(* CODESYS project AppSample_UDPCom_c550.project

Project tree, tasks and I/O mapping:
  c550_UDP_Example : Controller c550, Lenze, order no. FAST Runtime, version 1.11.0.21
      settings: 0x2001:0 = c550_UDP_Example; 0x2381:1 = 0; 0x2381:2 = 0; 0x2381:3 = 0; 0x2381:5 =                                 ; 0x2381:6 =                       ; 0x2381:7 =                 ; 0x2381:8 =                                                       ; 0x2451:1 = 0; 0x2451:2 = 0; 0x2451:3 = 0; 0x2451:4 = 0; 0x2459:1 = 0; 0x2459:2 = 0; 0x245A:2 = 0; 0x245A:3 = 0; 0x245A:4 = 0; 0x245A:5 = 0; 0x245B:1 = 2; 0x245C:1 = 52; 0x2471:13 = 100; 0x2471:14 = 100; 0x2471:51 = 1; 0x2471:103 = 6; 0x247B:1 = 0; 0x2859:1 = 2; 0x2859:2 = 0; 0x2859:3 = 2; 0x2859:4 = 2; 0x2859:5 = 2; 0x285A:1 = 0; 0x5820:1 = 2; 0x5851:31 = 100; 0x5910:1 = 0; 0x5910:2 = 0; 0x5910:3 = 0; 0x5910:4 = 0; 0x5910:5 = 0; 0x5910:6 = 0; 0x5910:7 = 0;
        0x5910:8 = 0; 0x5910:9 = 0; 0x5911:1 = 1; 0x5911:2 = 0; 0x5911:3 = 2; 0x5911:31 = 0; 0x5911:32 = 0; 0x5911:33 = 0; 0x5911:51 = 1; 0x5911:52 = 0; 0x5911:53 = 2; 0x5912:1 = 1; 0x5912:2 = 0; 0x5912:3 = 2; 0x5912:11 = 1; 0x5912:12 = 0; 0x5912:13 = 2; 0x5912:31 = 0; 0x5912:32 = 0; 0x5912:33 = 0; 0x5912:41 = 1; 0x5912:42 = 0; 0x5912:43 = 2; 0x5912:51 = 0; 0x5912:52 = 0; 0x5912:53 = 0; 0x5912:61 = 0; 0x5912:62 = 0; 0x5912:63 = 0; 0x5912:71 = 0; 0x5912:72 = 0; 0x5912:73 = 0; 0x5912:91 = 1; 0x5912:92 = 0; 0x5912:93 = 2; 0x5912:101 = 0; 0x5912:102 = 0; 0x5912:103 = 0; 0x5912:131 = 0; 0x5912:132 = 0;
        0x5912:133 = 0; 0x5912:151 = 0; 0x5912:152 = 0; 0x5912:153 = 0; 0x5913:1 = 0; 0x5913:2 = 0; 0x5913:3 = 0; 0x5913:7 = 0; 0x5913:8 = 50000; 0x5913:9 = 54999; 0x5913:10 = protocol name; 0x5913:11 = 0; 0x5913:12 = 0; 0x5913:13 = 0; 0x5913:17 = 0; 0x5913:18 = 50000; 0x5913:19 = 54999; 0x5913:20 = protocol name; 0x5913:21 = 0; 0x5913:22 = 0; 0x5913:23 = 0; 0x5913:27 = 0; 0x5913:28 = 50000; 0x5913:29 = 54999; 0x5913:30 = protocol name; 0x5913:31 = 0; 0x5913:32 = 0; 0x5913:33 = 0; 0x5913:37 = 0; 0x5913:38 = 50000; 0x5913:39 = 54999; 0x5913:40 = protocol name
    application Application
      libraries: CAA Types Extern, 3.5.17.0 (CAA Technical Workgroup); CAA Net Base Services, 3.5.17.0 (CAA Technical Workgroup); L_Util, 3.28.0.1 (Lenze); L_PLCLoggingAccess, 3.26.0.0 (Lenze); L_IE1P_ApplicationErrors, 3.30.0.53 (Lenze); L_MC2P_MotionControlCam, 3.30.0.17 (Lenze); L_SEMP_ErrorManagement, 3.26.0.0 (Lenze); L_IMHP_ModuleHandler, 3.30.0.11 (Lenze); L_IPAP_ParameterManagerAccess, 3.26.0.0 (Lenze); L_MC1P_MotionControlBasic, 3.30.0.173 (Lenze); L_SPMI_PlcParameterManager, 3.28.0.1 (Lenze); L_TB2P_TechModulesBasic, 3.30.0.61 (Lenze); L_TF2P_TechModulesFollowingPositioning, 3.30.0.62 (Lenze); L_TS2P_TechModulesSynchronizingCamming, 3.30.0.56 (Lenze); L_TW2P_TechModulesWindingTraversing, 3.30.0.7 (Lenze); L_TP2P_TechModulesProcessFunctions, 3.30.0.5 (Lenze); L_EtcSlaveConfig, 3.28.0.0 (Lenze); L_IC1P_ComponentDirectory, 3.30.0.8 (Lenze); L_ILMP_LicenseManager, 3.30.0.5 (Lenze); VisuDialogs, * (System)
      task MainTask (cyclic, interval t#5ms, priority 1, watchdog T#4ms x 1) calls MAIN_c550
      program MAIN_c550 [FBD]
      visualisation Visu_UDPCom_c550
      global variables GVL_ComponentHardware
      program GVL_ComponentHardwareCall [ST]
    I_O_Modul_Koppler : Coupler I/O moduls, Lenze, version 3.21.0.0
        settings: Group1 Task Name = 'MainTask'
        unmapped channels: Error, unused, unused, unused, unused, unused, unused, unused, ErrorID, AbsoluteCounter, unused, unused, unused, unused, unused, unused, unused, unused
    AxesGroups
    VirtualAxes
    ParameterEditor : Parameter Editor, Lenze, version 3.24.0.0
    FAST_System_Configuration : FAST System Configuration, Lenze, version 3.28.0.2
    FAST_System_Diagnosis : FAST System Diagnosis, Lenze, version 3.24.0.2
    OPC_UA : OPC UA Connectivity, Lenze, version 3.26.0.1
      UA_Server : OPC UA Server, Lenze, version 3.26.0.1
  text list GlobalTextList
  UDP_Com/
    function blocks/
      function block UDPCom [ST]: CreateCRC, Error, Peers, CheckIpIfBroadcastIsSet, RW
    data types/
      data type UDP_Telegram
    visualisation UDPCom_VISU
    internal/
      IpAddrHandling/
        visualisation IpAddrHandling_VISU
        FUNCTION/
          function Bytes4ToIpAddrString [ST]
          function IpAddressStringToBytes4 [ST]
        function block IpAddrHandling [ST]: CheckIpAddressSyntax
    text list NetBaseServices_ERROR
*)

// UDP_Com/data types/UDP_Telegram
{attribute 'pack_mode' := '0'}
TYPE UDP_Telegram :
STRUCT
	uiCRC: UINT; //Do not change this variable! Used for transferring the checksum!
	diUserData: DINT; //User data (can be of any type)
	//Add more user variables
END_STRUCT
END_TYPE

// c550_UDP_Example/Application/GVL_ComponentHardware
(* This code is generated automatically *)
(* Don't change the content! *)

{attribute 'qualified_only'}
{attribute 'linkalways'}
VAR_GLOBAL
	//Controller
	c550_UDP_Example 	: L_IC1P_ComponentHardware;

END_VAR

// c550_UDP_Example/Application/MAIN_c550
PROGRAM MAIN_c550
VAR
	fbUDPCom: UDPCom ;
	DataRead : UDP_Telegram;
	DataWrite: UDP_Telegram;
END_VAR

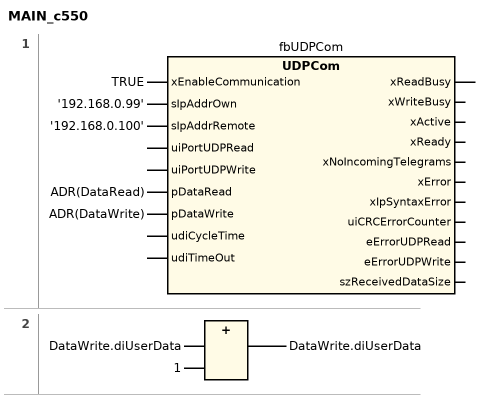
// NETWORK 1
fbUDPCom(
    xEnableCommunication := TRUE,
    sIpAddrOwn := '192.168.0.99',
    sIpAddrRemote := '192.168.0.100',
    pDataRead := ADR(DataRead),
    pDataWrite := ADR(DataWrite)); // UDPCom

// NETWORK 2
DataWrite.diUserData := DataWrite.diUserData + 1;

END_PROGRAM

// UDP_Com/function blocks/UDPCom
FUNCTION_BLOCK UDPCom
VAR_INPUT
	xEnableCommunication : BOOL;					 		  //Enabling UPD read or UPD write functions
	sIpAddrOwn			 : STRING[15];				 		  //IP address of this device
	sIpAddrRemote		 : STRING[15];				 		  //IP address of remote device
	uiPortUDPRead		 : UINT := 1240;			 		  //Port on this device via which UDP telegrams are received
	uiPortUDPWrite		 : UINT := 1241;			 		  //Port on this device via which UDP telegrams are transmitted
	pDataRead			 : POINTER TO UDP_Telegram; 		  //Passing the address of a variable of type UDP_Telegram. UDP_Telegram is a structure that contains the payload data for UDP communication
	pDataWrite			 : POINTER TO UDP_Telegram; 		  //Passing the address of a variable of type UDP_Telegram. UDP_Telegram is a structure that contains the payload data for UDP communication
	udiCycleTime		 : UDINT 					 := 100;  //Cycle time [ms] for sending UDP telegrams
	udiTimeOut			 : UDINT 					 := 2000; //Watchdog time, scaled in [ms]
END_VAR                                                   
VAR_OUTPUT                                                
	xReadBusy			 : BOOL;	   	//TRUE: Function block is busy in reading UDP data
	xWriteBusy			 : BOOL;	   	//TRUE: Function block is busy in writing UDP data
	xActive				 : BOOL;	   	//TRUE: Peers have opened for UDP communication on this device
	xReady				 : BOOL;	   	//TRUE: UDP data was read successfully
	xNoIncomingTelegrams : BOOL;	   	//TRUE: No handshake telegram has been received within the watchdog time period (udiTimeOut)
	xError				 : BOOL;	   	//TRUE: An error has occured during function block execution (for more details please refer to status output eError)
	xIpSyntaxError    	 : BOOL;	   	//TRUE: The IP address set in sIpAddrOwn and/or in sIpAddrRemote has an incorrect syntax
	uiCRCErrorCounter	 : UINT;		//If the checksum check detects incorrect data in the received telegram, uiCRCErrorCounter is incremented
	eErrorUDPRead    	 : CAA.ERROR; 	//Error number for the UDP read process, in the case of xError = TRUE
	eErrorUDPWrite	  	 : CAA.ERROR;	//Error number for the UDP write process, in the case of xError = TRUE
	szReceivedDataSize	 : CAA.SIZE;  	//Size in bytes of the received data
END_VAR
VAR
	(* FB instances *)
	fbIpAddrHandlingOwn	   : IpAddrHandling;	//Function block for IP-Address handling
	fbIpAddrHandlingRemote : IpAddrHandling;   	//Function block for IP-Address handling 	
	fbPeerRX			   : NBS.UDP_Peer;		//Function block to open a peer to read UDP telegrams on function block UDP_Receive1
	fbPeerTX			   : NBS.UDP_Peer;		//Function block to open a peer to transmit UDP telegram on function block UDP_Send1
	fbUDPReceive		   : NBS.UDP_Receive;	//Function block for reading UDP data via peer 1
	fbUDPSend			   : NBS.UDP_Send;		//Function block for transmitting UDP telegram on peer 2
	fbTrigWatchdogTimer	   : R_TRIG;    		//Edge detection to start the watchdog timer		 
	fbWatchdogTimer		   : TON;				//Timer function block for watchdog evaluation
	fbTimerCyclic		   : TON;				//Timer function block for cyclic data transmission
	
	(*Internal variables *)
	xReadActive    	: BOOL;
	xWriteActive 	: BOOL;
	szSizeDataRead 	: CAA.SIZE;
	szSizeDataWrite : CAA.SIZE;
	xBroadcastIsSet : BOOL;
	uiCRC: UINT; //CRC
END_VAR

(* Calling the block instances of IpAddrHandling ====================================================*)
fbIpAddrHandlingOwn(psIpAddrIN 		:= ADR(sIpAddrOwn));
fbIpAddrHandlingRemote(psIpAddrIN 	:= ADR(sIpAddrRemote));

xBroadcastIsSet := CheckIpIfBroadcastIsSet(sIpAddrString := sIpAddrRemote);

(* Set xIpSyntaxError ===============================================================================*)
IF fbIpAddrHandlingOwn.xIpSyntaxError OR fbIpAddrHandlingRemote.xIpSyntaxError THEN
	xIpSyntaxError := TRUE;
ELSE
	xIpSyntaxError := FALSE;
END_IF

(* Get the number of bytes of user data by dereferencing the pointer ================================*)
szSizeDataRead := SIZEOF(pDataRead^);
szSizeDataWrite := SIZEOF(pDataWrite^);

(* UDP peers ========================================================================================*)
Peers();

(* UDP read write ===================================================================================*)
RW();

(* Set errors =======================================================================================*)
Error();

(* Set output variables =============================================================================*)
xActive := xReadActive AND xWriteActive;

(* Create a simple checksum by adding a maximum of 128 byte packets *)
METHOD PRIVATE CreateCRC : UINT
VAR_INPUT
	pData: POINTER TO UDP_Telegram;
END_VAR
VAR
	paby	: POINTER TO ARRAY[0..130] OF BYTE;
	uiSize	: UINT;
	ui 		: UINT := 2;
END_VAR

paby := pData;
uiSize := SIZEOF(pData^) - 2;
IF uiSize >= 128 THEN
	uiSize := 128;
END_IF

FOR ui := 2 TO uiSize BY 1 DO
	CreateCRC := CreateCRC + paby^[ui];
END_FOR
END_METHOD

ACTION Error:
(* Set errors =======================================================================================*)

xError := fbPeerRX.xError OR fbUDPReceive.xError OR fbPeerTX.xError OR fbUDPSend.xError;

IF fbPeerRX.xError THEN        
	eErrorUDPRead := fbPeerRX.eError;
ELSIF fbUDPReceive.xError THEN  
	eErrorUDPRead := fbUDPReceive.eError;
ELSE                                
	eErrorUDPRead := 0;
END_IF

IF fbPeerTX.xError THEN
	eErrorUDPWrite := fbPeerTX.eError;
ELSIF fbUDPSend.xError THEN
	eErrorUDPWrite := fbUDPSend.eError;
ELSE
	eErrorUDPWrite := 0;
END_IF
END_ACTION

ACTION Peers:
(* READ | Open a peer to read data from remote IP address============================================*)
//Change IP-Address setting if an broadcast IP is set
IF xBroadcastIsSet THEN
	fbPeerRX.ipAddr.sAddr := sIpAddrRemote;	//setting remote IP address (access of element of structure NBS.IP_ADDR)
ELSE
	fbPeerRX.ipAddr.sAddr := sIpAddrOwn; 	//setting own IP address (access of element of structure NBS.IP_ADDR)
END_IF

//Open a peer for receive Data
fbPeerRX(xEnable := xEnableCommunication, uiPort := uiPortUDPRead);

//Set xReadActive if the peer opened successfully
xReadActive := fbPeerRX.xActive AND fbPeerRX.hPeer<>0;


(* WRITE | Open a peer to transmit data to remote IP address=========================================*)
//Open a peer for transmit Data
fbPeerTX.ipAddr.sAddr := sIpAddrOwn; // setting own IP address (access of element of structure NBS.IP_ADDR)
fbPeerTX(xEnable := xEnableCommunication, uiPort := uiPortUDPWrite);

//Set xWriteActive if the peer opened successfully
xWriteActive := fbPeerTX.xActive AND fbPeerTX.hPeer<>0;
END_ACTION

(* Check whether the last octet in the IP address is set to 255 (broadcast) *)
METHOD PRIVATE CheckIpIfBroadcastIsSet : BOOL
VAR_INPUT
	sIpAddrString: STRING[15];
END_VAR
VAR
	usiStringLengh: USINT;
	sTemp: STRING[4];
END_VAR

usiStringLengh := TO_USINT(LEN(sIpAddrString));
sTemp := MID(sIpAddrString, 4, usiStringLengh - 3);

IF sTemp = '.255' THEN
	CheckIpIfBroadcastIsSet := TRUE;
ELSE
	CheckIpIfBroadcastIsSet := FALSE;
END_IF
END_METHOD

ACTION RW:

(* READ =============================================================================================*)
//UDP receive
fbUDPReceive(xEnable := xReadActive,
			 hPeer	 := fbPeerRX.hPeer,
			 szSize	 := szSizeDataRead,
			 pData	 := pDataRead,
			 xDone	 => ,
			 xBusy	 => xReadBusy,
			 xReady	 => xReady);

//CRC check
	uiCRC := CreateCRC(pData := pDataRead);
	IF uiCRC <> pDataRead^.uiCRC THEN
		uiCRCErrorCounter := uiCRCErrorCounter + 1;
	ELSIF xEnableCommunication = FALSE THEN
		uiCRCErrorCounter := 0;
	END_IF
	
//Get number of bytes received from the sender
IF fbUDPReceive.xReady OR NOT xReadActive THEN
	szReceivedDataSize := fbUDPReceive.szCount; 
END_IF

//Generation of watchdog alert
fbTrigWatchdogTimer(CLK	:= xReady);
fbWatchdogTimer(IN	:= xReadActive AND NOT fbTrigWatchdogTimer.Q AND (udiTimeOut<>0),
				PT	:= UDINT_TO_TIME(udiTimeOut),
				Q	=> xNoIncomingTelegrams);

(* WRITE ============================================================================================*)
//Logic for cyclic transmission
fbTimerCyclic(IN := NOT fbTimerCyclic.Q, PT	:= UDINT_TO_TIME(LIMIT(9,udiCycleTime-1,4294967294))); 

//Execute UDP transmission
fbUDPSend.xExecute := xWriteActive AND (udiCycleTime > 0 AND fbTimerCyclic.Q); 

//Create CRC
IF fbUDPSend.xExecute THEN
	pDataWrite^.uiCRC := CreateCRC(pData := pDataWrite);
END_IF

//UDP send
fbUDPSend.ipAddr.sAddr	:= sIpAddrRemote; 
fbUDPSend(	hPeer 	:= fbPeerTX.hPeer,
			uiPort	:= uiPortUDPWrite,
			szSize	:= szSizeDataWrite,
			pData	:= pDataWrite,	
			xDone	=> ,				
			xBusy	=> );
END_ACTION

END_FUNCTION_BLOCK

// UDP_Com/internal/IpAddrHandling/IpAddrHandling
(*	This function block is responsible for setting an IP address. This can be changed in two places:												*)
(*		1. In a user-created variable of type STRING[15]. To do this, 																				*)
(*		   the address of this variable must be transferred to the function block input “psIpAddrIN”.												*)
(*		2. In the visualization "IpAddrHandling_VISU" available for this function block.															*)
(*																																					*)
(*	If the address is changed with correct syntax in one of these two places, it is output in "sIpAddrOut". If the user variable, which is passed  	*)
(*	as a pointer to "psIpAddrIN", is written cyclically in the PLC program with a syntactically correct IP address, this is always output to 		*)
(*	"sIpAddrOut". A change via the visualization is then no longer possible. 																		*)															
FUNCTION_BLOCK IpAddrHandling
VAR_INPUT
	psIpAddrIN: POINTER TO STRING[15];
END_VAR
VAR_OUTPUT
	sIpAddrOut: STRING(15);
	xIpSyntaxError: BOOL;
END_VAR
VAR
	sIpAddrIN: STRING[15];
	sIpAddrVisu: STRING[15];
	abyIpVISU: ARRAY[0..3] OF BYTE := [192, 168, 5, 99];
	
	sIpAddrInOLD: STRING[15];
	sIpAddrVisuOLD: STRING[15] := '0.0.0.0';
	
	xChangeDetected : BOOL;
	xCheckInput: BOOL;
	usiStep: USINT;
END_VAR


sIpAddrVisu := Bytes4ToIpAddrString(abyIpVISU);

IF psIpAddrIN <> 0 THEN
	sIpAddrIN := psIpAddrIN^;
END_IF
	
CASE usiStep OF

	00: //Check for changes
	
		IF sIpAddrIN <> sIpAddrInOLD THEN //Check whether the set IP address in sIpAddrIN has changed

			IF CheckIpAddressSyntax(sIpAddrString := sIpAddrIN) THEN
				xIpSyntaxError := FALSE;
				usiStep := 10; //Next step
			ELSE
				sIpAddrInOLD := sIpAddrIN;
				xIpSyntaxError := TRUE;
			END_IF
			
		ELSIF sIpAddrVisu <> sIpAddrVisuOLD THEN //Check whether the IP address set in sIpAddrVisu has changed
			psIpAddrIN^ := sIpAddrVisu;
			usiStep := 10; //Next step
		END_IF
	
	10: //Write output
	
		IF CheckIpAddressSyntax(sIpAddrString := sIpAddrIN) = FALSE THEN
			xIpSyntaxError := TRUE;
		ELSE
			xIpSyntaxError := FALSE;
		END_IF
	
		IF (sIpAddrIN = sIpAddrVisu) OR xIpSyntaxError THEN
			sIpAddrVisuOLD 	:= sIpAddrVisu;
			sIpAddrInOLD 	:= sIpAddrVisu;
			sIpAddrOut 		:= sIpAddrVisu;
		ELSE 
			sIpAddrInOLD	:= sIpAddrIN;
			sIpAddrVisuOLD 	:= sIpAddrIN;
			sIpAddrOut 		:= sIpAddrIN;
		END_IF
		
		abyIpVISU := IpAddressStringToBytes4(sIpAddrOut); //Write the output back to Visu
		
		usiStep := 00;

END_CASE

METHOD PRIVATE CheckIpAddressSyntax : BOOL //TRUE: Syntax correct | FALSE: Syntax not correct
VAR_INPUT
	sIpAddrString: STRING[15];
END_VAR
VAR
	usiStringLengh: USINT;
	i: USINT;
	j: USINT;
	sTemp: STRING[1];
	
	sTemp_j: STRING[1];
	
	usiDotCounter: USINT;
	usiSymbolCounterTemp: USINT;
	usiSymbolCounterTotal: USINT;
END_VAR

usiSymbolCounterTemp := 0;
usiSymbolCounterTotal := 0;
usiDotCounter := 0;

usiStringLengh := TO_USINT(LEN(sIpAddrString));

FOR i := 1 TO (usiStringLengh) BY 1 DO
	
	sTemp := MID(sIpAddrString, 1, i);
	
	FOR j := 0 TO 9 BY 1 DO
		sTemp_j := TO_STRING(j);
		IF (usiSymbolCounterTemp >= 0 AND usiSymbolCounterTemp <= 2) AND sTemp = sTemp_j THEN
			usiSymbolCounterTotal := usiSymbolCounterTotal + 1;
			usiSymbolCounterTemp := usiSymbolCounterTemp + 1;
			EXIT;
		ELSIF (usiSymbolCounterTemp >= 1 AND usiSymbolCounterTemp <= 3) AND sTemp = '.' THEN
			usiSymbolCounterTotal := usiSymbolCounterTotal + 1;
			usiSymbolCounterTemp := 0;
			usiDotCounter := usiDotCounter + 1;
			EXIT;
		END_IF
	END_FOR

END_FOR

IF usiStringLengh = usiSymbolCounterTotal AND usiDotCounter = 3 THEN
	CheckIpAddressSyntax := TRUE;
ELSE
	CheckIpAddressSyntax := FALSE;
END_IF
END_METHOD

END_FUNCTION_BLOCK

// UDP_Com/internal/IpAddrHandling/FUNCTION/Bytes4ToIpAddrString
{attribute 'hide_all_locals'}
FUNCTION Bytes4ToIpAddrString : STRING(15)
VAR_INPUT
	abyIPAddress: ARRAY[0..3] OF BYTE;
END_VAR
VAR
	sTemp: STRING(15);
END_VAR


sTemp := CONCAT(TO_STRING(abyIPAddress[0]), '.');
sTemp := CONCAT(sTemp, TO_STRING(abyIPAddress[1]));
sTemp := CONCAT(sTemp, '.');
sTemp := CONCAT(sTemp, TO_STRING(abyIPAddress[2]));
sTemp := CONCAT(sTemp, '.');
sTemp := CONCAT(sTemp, TO_STRING(abyIPAddress[3]));

Bytes4ToIpAddrString := sTemp;

END_FUNCTION

// UDP_Com/internal/IpAddrHandling/FUNCTION/IpAddressStringToBytes4
FUNCTION IpAddressStringToBytes4 : ARRAY[0..3] OF BYTE
VAR_INPUT
	sIpAddrString: STRING[15];
END_VAR
VAR
	iNumberOfDecimals_1: INT;
	iNumberOfDecimals_2: INT;
	iNumberOfDecimals_3: INT;

	sTemp2: STRING[15];
	sTemp3: STRING[15];
	sTemp4: STRING[15];
END_VAR


//First octet
iNumberOfDecimals_1 := FIND(sIpAddrString, '.');
IpAddressStringToBytes4[0] := TO_BYTE(MID(sIpAddrString, iNumberOfDecimals_1 -1, 1));
sTemp2 := DELETE(sIpAddrString, iNumberOfDecimals_1, 1);

//Second octet
iNumberOfDecimals_2 := FIND(sTemp2, '.');
IpAddressStringToBytes4[1] := TO_BYTE(MID(sTemp2, iNumberOfDecimals_2 -1, 1));
sTemp3 := DELETE(sTemp2, iNumberOfDecimals_2, 1);

//Third octet
iNumberOfDecimals_3 := FIND(sTemp3, '.');
IpAddressStringToBytes4[2] := TO_BYTE(MID(sTemp3, iNumberOfDecimals_3 -1, 1));
sTemp4 := DELETE(sTemp3, iNumberOfDecimals_3, 1);

//Fourth octet
IpAddressStringToBytes4[3] := TO_BYTE(sTemp4);

END_FUNCTION

// c550_UDP_Example/Application/GVL_ComponentHardwareCall
{attribute 'linkalways'}
PROGRAM GVL_ComponentHardwareCall
VAR
END_VAR

(* This code is generated automatically *)
(* Don't change the content! *)

//Controller
GVL_ComponentHardware.c550_UDP_Example();

END_PROGRAM

// UDP_Com/UDPCom_VISU
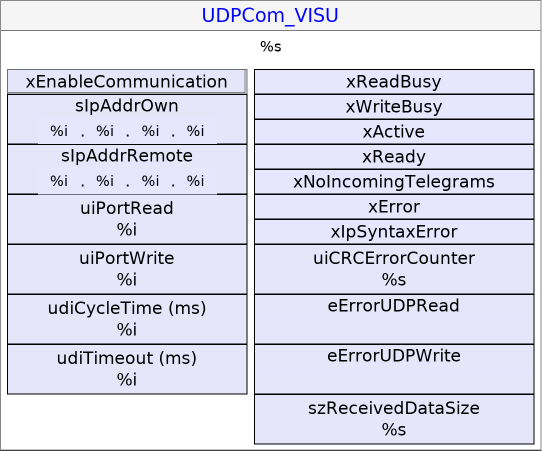
VISUALIZATION UDPCom_VISU  // 542x451
VAR_INPUT
	{attribute 'parameterstringof' := 'm_Input_FB'}
	m_Input_INST_Str : STRING;
END_VAR
VAR_IN_OUT
	m_Input_FB: UDPCom;
END_VAR
    Rectangle (0,0 541x451)
    Rectangle (254,194 280x25), "xError", colour toggle: m_Input_FB.xError
    Button (7,69 240x25), "xEnableCommunication", colour toggle: m_Input_FB.xEnableCommunication
        toggle m_Input_FB.xEnableCommunication
    Rectangle (7,194 240x50), "uiPortRead %i", text variable: m_Input_FB.uiPortUDPRead
        OnMouseClick: write the text variable via Default
    Rectangle (7,344 240x50), "udiTimeout (ms) %i", text variable: m_Input_FB.udiTimeout
        OnMouseClick: write the text variable via Default
    Rectangle (0,0 541x31), "UDPCom_VISU"
    Textfield (0,31 542x31), "%s", text variable: m_Input_INST_Str
    Rectangle (254,169 280x25), "xNoIncomingTelegrams", colour toggle: m_Input_FB.xNoIncomingTelegrams
    Rectangle (254,144 280x25), "xReady", colour toggle: m_Input_FB.xReady
    Rectangle (254,119 280x25), "xActive", colour toggle: m_Input_FB.xActive
    Rectangle (254,69 280x25), "xReadBusy", colour toggle: m_Input_FB.xReadBusy
    Rectangle (254,394 280x50), "szReceivedDataSize %s", text variable: m_Input_FB.szReceivedDataSize
    Group (7,94 240x50)
        Rectangle (0,0 240x50), "sIpAddrOwn"
        Frame (31,24 179x26)
            shows IpAddrHandling_VISU(m_Input_FB := m_Input_FB.fbIpAddrHandlingOwn)
    Group (7,144 240x50)
        Rectangle (0,0 240x50), "sIpAddrRemote"
        Frame (31,24 179x26)
            shows IpAddrHandling_VISU(m_Input_FB := m_Input_FB.fbIpAddrHandlingRemote)
    Rectangle (7,294 240x50), "udiCycleTime (ms) %i", text variable: m_Input_FB.udiCycleTime
        OnMouseClick: write the text variable via Default
    Rectangle (254,219 280x25), "xIpSyntaxError", colour toggle: m_Input_FB.xIpSyntaxError
    Group (254,294 280x50)
        Rectangle (0,0 280x50), "eErrorUDPRead"
        Rectangle (1,24 278x25), text list: 'NetBaseServices_ERROR', text index: m_Input_FB.eErrorUDPRead
    Rectangle (7,244 240x50), "uiPortWrite %i", text variable: m_Input_FB.uiPortUDPWrite
        OnMouseClick: write the text variable via Default
    Group (254,344 280x50)
        Rectangle (0,0 280x50), "eErrorUDPWrite"
        Rectangle (1,24 278x25), text list: 'NetBaseServices_ERROR', text index: m_Input_FB.eErrorUDPWrite
    Rectangle (254,94 280x25), "xWriteBusy", colour toggle: m_Input_FB.xWriteBusy
    Rectangle (254,244 280x50), "uiCRCErrorCounter %s", text variable: m_Input_FB.uiCRCErrorCounter
END_VISUALIZATION

// UDP_Com/internal/IpAddrHandling/IpAddrHandling_VISU
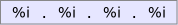
VISUALIZATION IpAddrHandling_VISU  // 178x25
VAR_IN_OUT
	m_Input_FB: IpAddrHandling;
END_VAR
    Rectangle (0,0 178x25)
    Rectangle (0,0 42x25), "%i", text variable: m_Input_FB.abyIpVISU[0]
        OnMouseClick: write the text variable via Default
    Rectangle (46,0 42x25), "%i", text variable: m_Input_FB.abyIpVISU[1]
        OnMouseClick: write the text variable via Default
    Rectangle (91,0 42x25), "%i", text variable: m_Input_FB.abyIpVISU[2]
        OnMouseClick: write the text variable via Default
    Rectangle (136,0 42x25), "%i", text variable: m_Input_FB.abyIpVISU[3]
        OnMouseClick: write the text variable via Default
    Label (131,0 7x24), "."
    Label (86,0 7x24), "."
    Label (41,0 7x24), "."
END_VISUALIZATION

// c550_UDP_Example/Application/Visu_UDPCom_c550
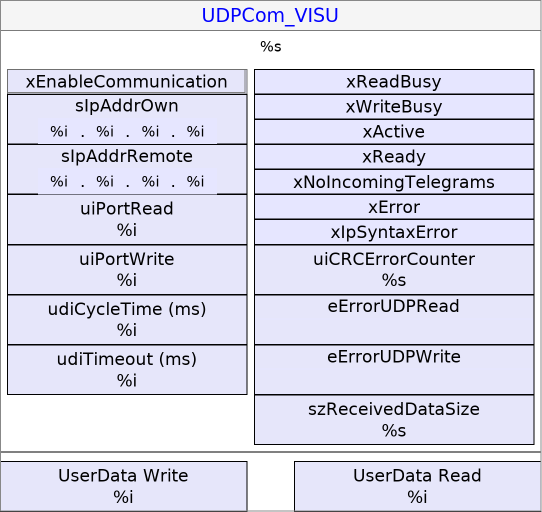
VISUALIZATION Visu_UDPCom_c550  // 542x512
    Rectangle (0,461 247x51), "UserData Write %i", text variable: MAIN_c550.DataWrite.diUserData
        OnMouseClick: write the text variable via Default
    Rectangle (294,461 247x51), "UserData Read %i", text variable: MAIN_c550.DataRead.diUserData
        OnMouseClick: write the text variable via Default
    Frame (0,0 542x452)
        shows UDPCom_VISU(m_Input_FB := MAIN_c550.fbUDPCom)
END_VISUALIZATION

(* text list NetBaseServices_ERROR (id | default)
  0 | NO_ERROR
  6000 | FIRST_ERROR
  6001 | TIME_OUT
  6002 | INVALID_ADDR
  6003 | INVALID_HANDLE
  6004 | INVALID_DATAPOINTER
  6005 | INVALID_DATASIZE
  6006 | UDP_RECEIVE_ERROR
  6007 | UDP_SEND_ERROR
  6008 | UDP_SEND_NOT_COMPLETE
  6009 | UDP_OPEN_ERROR
  6010 | UDP_CLOSE_ERROR
  6011 | TCP_SEND_ERROR
  6012 | TCP_RECEIVE_ERROR
  6013 | TCP_OPEN_ERROR
  6014 | TCP_CONNECT_ERROR
  6015 | TCP_CLOSE_ERROR
  6016 | TCP_SERVER_ERROR
  6017 | WRONG_PARAMETER
  6018 | ERROR_UNKNOWN
  6019 | TCP_NO_CONNECTION
  6020 | IOCTL_ERROR
  6050 | FIRST_MF
  6099 | LAST_ERROR
   |  *)
